FUNCTION_BLOCK FB_Downtime_LOG
VAR_INPUT
	CansCounter: REAL;
	RealDowntimeConditions: BOOL;
	FillerRoom: STRING;
	Start_buttonHMI: BOOL;
	End_buttonHMI: BOOL;
	ID_StopReason: INT; 
	Confirm_buttonHMI: BOOL;
	
END_VAR
VAR_OUTPUT
	ProductionRunning: BOOL;
	ValidStop: BOOL; //DowntimeLog: BOOL;
	CODE_DowntimeLog: STRING;
	Downtime_View_Control: BOOL;
	LineStopsCounter: INT;
	
	
END_VAR
VAR
	FixedSchedule_Verify: FixedSchedule_FillerRoom;
	onSchedule: BOOL;
	StartButton: R_TRIG;
	RedCan_Button: R_TRIG;
	
	StartedCounter: BOOL;
	RS_Dowtime: RS;
	Reset_DowntimeLog: BOOL;
	DT_Confirm_Button: R_TRIG;
	DT_ConfirmB: BOOL;
	
 	RealStop: BOOL;
	
	ValidStop_Verifier: TON;
	PulseHMI_StopScreen: TP;
	Codes_StopReason_HMI: Codes_StopReason;
	VALID_StopCode: BOOL;
	SaveStopReasonsValues: R_TRIG;
	StopNumber: INT;	
	FillerStopped: CTU; //Counter stops
	CansDetected: R_TRIG;
END_VAR

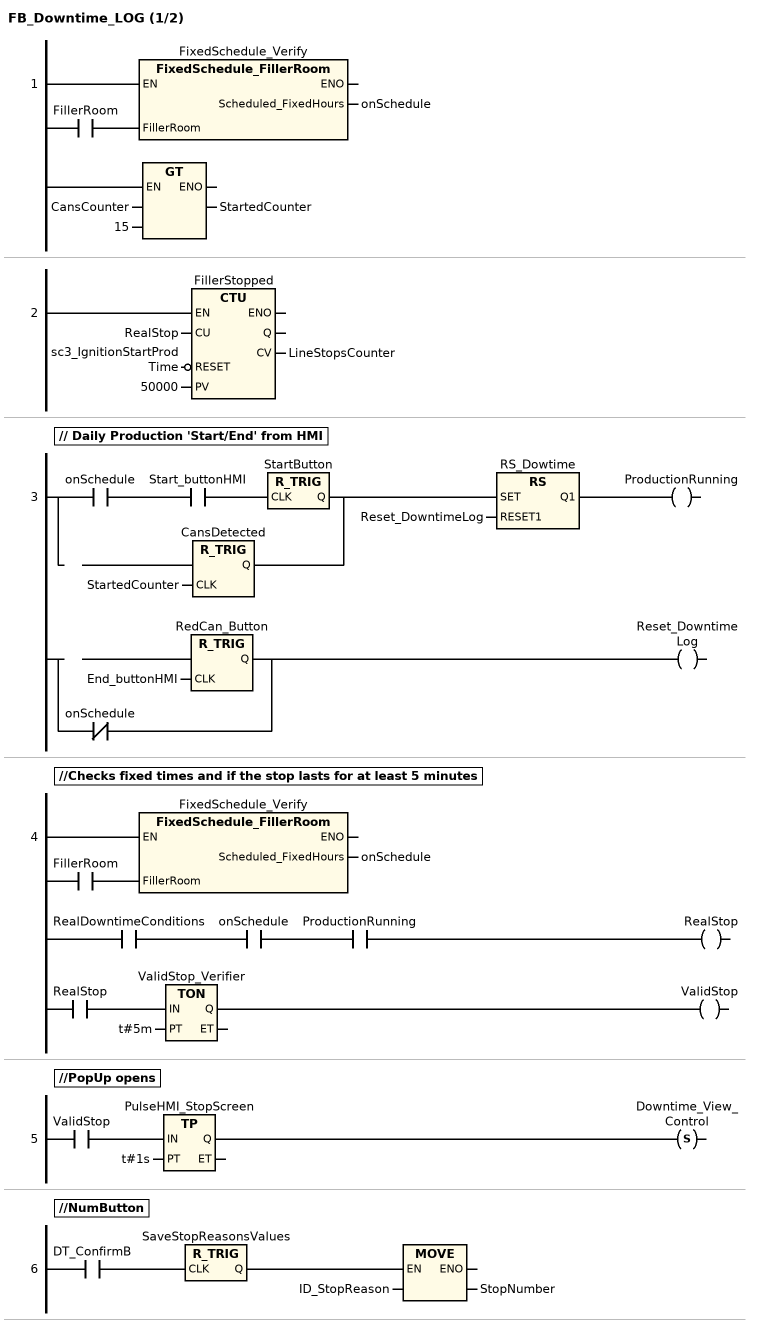
// NETWORK 1
FixedSchedule_Verify(FillerRoom := FillerRoom, Scheduled_FixedHours => onSchedule); // FixedSchedule_FillerRoom
StartedCounter := CansCounter > 15;

// NETWORK 2
FillerStopped(CU := RealStop, RESET := NOT sc3_IgnitionStartProdTime, PV := 50000, CV => LineStopsCounter); // CTU

// NETWORK 3
// label: // Daily Production 'Start/End' from HMI
StartButton(CLK := onSchedule AND Start_buttonHMI); // R_TRIG
CansDetected(CLK := StartedCounter); // R_TRIG
RS_Dowtime(SET := StartButton.Q OR CansDetected.Q, RESET1 := Reset_DowntimeLog); // RS
ProductionRunning := RS_Dowtime.Q1;
RedCan_Button(CLK := End_buttonHMI); // R_TRIG
Reset_DowntimeLog := RedCan_Button.Q OR NOT onSchedule;

// NETWORK 4
// label: //Checks fixed times and if the stop lasts for at least 5 minutes
FixedSchedule_Verify(FillerRoom := FillerRoom, Scheduled_FixedHours => onSchedule); // FixedSchedule_FillerRoom
RealStop := (RealDowntimeConditions AND onSchedule) AND ProductionRunning;
ValidStop_Verifier(IN := RealStop, PT := t#5m); // TON
ValidStop := ValidStop_Verifier.Q;

// NETWORK 5
// label: //PopUp opens
PulseHMI_StopScreen(IN := ValidStop, PT := t#1s); // TP
Downtime_View_Control S= PulseHMI_StopScreen.Q;

// NETWORK 6
// label: //NumButton
SaveStopReasonsValues(CLK := DT_ConfirmB); // R_TRIG
IF SaveStopReasonsValues.Q THEN StopNumber := ID_StopReason; END_IF

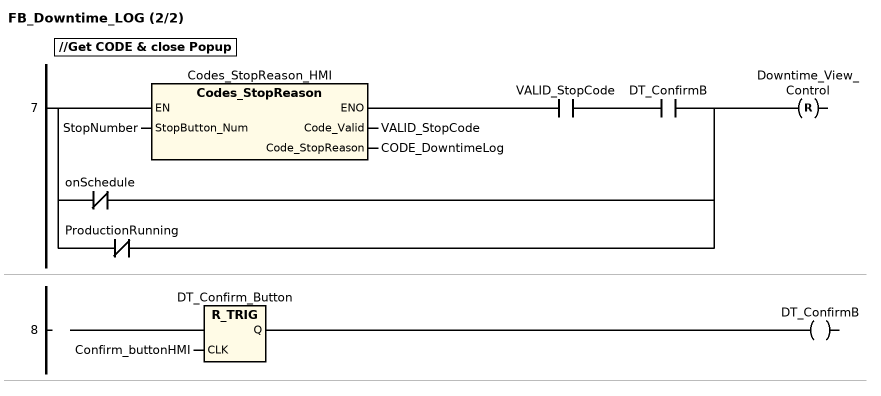
// NETWORK 7
// label: //Get CODE & close Popup
Codes_StopReason_HMI(
    EN := TRUE,
    StopButton_Num := StopNumber,
    Code_Valid => VALID_StopCode,
    Code_StopReason => CODE_DowntimeLog); // Codes_StopReason
Downtime_View_Control R= TRUE AND VALID_StopCode AND DT_ConfirmB OR NOT onSchedule OR NOT ProductionRunning;

// NETWORK 8
DT_Confirm_Button(CLK := Confirm_buttonHMI); // R_TRIG
DT_ConfirmB := DT_Confirm_Button.Q;

END_FUNCTION_BLOCK

(* stored: Version 1.1.0.1, ProductVersion 3.1.4024.15
   POU FB_Downtime_LOG: Id {b101b8dc-09d0-4371-8831-1b83bc40896f}, SpecialFunc None *)
